INTERFACE I_Datatype extends I_Serializable, I_Deserializable, I_Disposable

PROPERTY PUBLIC Address : PVOID
GET
END_GET
END_PROPERTY

METHOD PUBLIC ClearReference
VAR_INPUT
END_VAR
END_METHOD

PROPERTY PUBLIC Identifier : T_MAXSTRING
GET
END_GET
END_PROPERTY

METHOD PUBLIC SerializeTypeWith
VAR_INPUT
	Serializer : I_Serializer;
END_VAR
END_METHOD

PROPERTY PUBLIC Size : UDINT
GET
END_GET
END_PROPERTY

METHOD TryMakeReferenceOf : BOOL
VAR_INPUT
	Target : I_Datatype;
END_VAR
END_METHOD

END_INTERFACE

(* stored: Version 1.1.0.1, ProductVersion 3.1.4024.12
   Itf I_Datatype: Id {60a3fa78-0098-0a1a-3ab1-3b6b68cfc3f8}
   Property Address: Id {97ce40cf-daf1-4f84-befc-3d953dbd0739}
   Get Get: Id {cbd086cf-89d8-45a8-89c5-e52e3a096e7d}
   Method ClearReference: Id {d6ba8507-aaaa-0d79-12ee-6da70653c60f}
   Property Identifier: Id {b5ede973-026a-40e2-b656-ccf5a34daaf0}
   Get Get: Id {bd9a47c5-8817-48b1-a2cd-e41da6b3e2dd}
   Method SerializeTypeWith: Id {62fe74e3-7708-080e-2978-6b48ab2638bd}
   Property Size: Id {5c04081a-bb6e-4218-8597-9b7757149fa1}
   Get Get: Id {fdc689ce-7c38-465d-a111-883a520bad02}
   Method TryMakeReferenceOf: Id {baec0ebb-3447-0677-3e86-cc7b3c3ce04c} *)
